TYPE AxesDeltaUnits :
(
	DEGREES := 0,
	RADIANS := 1
);
END_TYPE

(* stored: Version 1.1.0.1, ProductVersion 3.1.4019.2
   DUT AxesDeltaUnits: Id {d383a3a4-a30d-4aed-a52f-ae3b7f19ae20} *)
